Staubli VAL3: getFrame.pgx

public program getFrame(string& x_sFrm, frame& x_fFrame)
begin
  x_sFrm=sFrameName
  x_fFrame.trsf=fFrame[sFrameName].trsf
end
